PROGRAM prgDataGrab
VAR
	tGrabData: BOOL;
	
	DataIndex: ULINT;
	MaxAxisGrab: ULINT;
	tAxisFull: BOOL;
	
	visuBoxControl1:FB_BoxControl;
	visuBoxControl2:FB_BoxControl;
	visuBoxControl3:FB_BoxControl;
	
	CheckWindow1:FB_Window;
	
END_VAR

actPopulateAxis();


//temp control boxes
//change the button control function on the boxes
visuBoxControl1(iqBoxdata := dataGrab.dataCurrentVisu.box1);
visuBoxControl2(iqBoxdata := dataGrab.dataCurrentVisu.box2);
visuBoxControl3(iqBoxdata := dataGrab.dataCurrentVisu.box3);


CheckWindow1(	dataAxis		:=	dataGrab.dataCurrentVisu.axis,
				i1				:=	datagrab.dataCurrentVisu.box1.i1, //co-ords
				i2				:=	datagrab.dataCurrentVisu.box1.i2, //co-ords
				i3				:=	datagrab.dataCurrentVisu.box1.i3, //co-ords
				i4				:=	datagrab.dataCurrentVisu.box1.i4, //co-ords
				LeftPermSide	:=	datagrab.dataCurrentVisu.box1.leftStatus,
				RightPermSide	:=	datagrab.dataCurrentVisu.box1.rightStatus,
				TopPermSide		:=	datagrab.dataCurrentVisu.box1.topStatus,
				BottomPermSide	:=	datagrab.dataCurrentVisu.box1.bottomStatus
				);

ACTION actPopulateAxis:
MaxAxisGrab := 100;

//populate axis

(*
IF tGrabData THEN

DataIndex := DataIndex + 1;

	//lets grab data
	IF DataIndex < MaxAxisGrab THEN
		dataGrab.axis1.grabTime[dataIndex] := DataIndex;
		dataGrab.axis1.grabData[dataIndex] := 123.456;
		
		
	END_IF
	
	IF DataIndex >= MaxAxisGrab THEN
		tAxisFull := TRUE;
		tGrabData := FALSE;
	END_IF
	

END_IF


*)
END_ACTION

END_PROGRAM

(* stored: Version 1.1.0.1, ProductVersion 3.1.4024.11
   POU prgDataGrab: Id {2109d875-92f9-03a8-2fd3-97b38c500296}, SpecialFunc None
   Action actPopulateAxis: Id {17e9635a-4bdc-076c-0e86-b67297dd33f3} *)
